# EPICS autosave request: iocBoot/sioc-li21-bl01/blen_manual.req
file "manual.req" AREA=LI21,POS=266,INST=BL11A
file "manual.req" AREA=LI21,POS=266,INST=BL11B
